// This function has been automatically generated from the project information.
{attribute 'signature_flag' := '1073741824'}
{attribute 'TcGenerated'}
{attribute 'no-analysis'}
FUNCTION F_GetTitle : WSTRING
VAR_INPUT
	
END_VAR

F_GetTitle := "ScalingAndConversion";

END_FUNCTION

(* stored: Version 1.1.0.1
   POU F_GetTitle: Id {c4e1bbfd-c390-4010-8fb0-c050326c6720}, SpecialFunc None *)
